# EPICS autosave request: CARSApp/Db/newport_table_settings.req
# FILE... newport_table_settings.req
$(P)$(T)lx
$(P)$(T)lz
$(P)$(T)D0x
$(P)$(T)D0y
$(P)$(T)D0z
$(P)$(T)d1
$(P)$(T)d2
$(P)$(PM4):Readback
$(P)$(PM5):Readback
$(P)$(PM6):Readback
$(P)$(PM7):Readback
$(P)$(PM8):Readback
